// TIA Portal V16 export
// export: Created 2024-12-03T15:41:45.2417545Z, ExportSetting WithReadOnly, DisplayName Totally Integrated Automation Portal, DisplayVersion V16 Update 6, DisplayName TIA Portal Version Control Interface, DisplayVersion V16 Update 2, DisplayName TIA Portal Openness, DisplayVersion V16 Update 6, DisplayName TIA Portal Teamcenter Gateway, DisplayVersion V16, DisplayName SINAMICS Startdrive Advanced, DisplayVersion V16 Update 5, DisplayName SINAMICS Startdrive G130, G150, S120, S150, SINAMICS MV, S210, DisplayVersion V16 Update 5, DisplayName SINAMICS Startdrive G110M, G120, G120C, G120D, G120P, G115D, DisplayVersion V16 Update 5, DisplayName STEP 7 Professional, DisplayVersion V16 Update 6, DisplayName STEP 7 Safety, DisplayVersion V16, DisplayName WinCC Advanced / Unified PC, DisplayVersion V16 Update 6
TYPE "I_ScaleDataUdt"
// stored: CreationDate 2023-08-01T06:41:33.0989412Z, InterfaceModifiedDate 2023-08-01T07:53:02.5904875Z, IsConsistent true, LibraryConformanceStatus The object is library-conformant., ModifiedDate 2023-08-01T07:53:02.5904875Z
   STRUCT
      grossWeight : DInt;
      netWeight : DInt;
      inputStatus : Word;
      commandStatus : Word;
      outputStatus : Word;
   END_STRUCT;
END_TYPE
